PROGRAM MAIN
VAR
END_VAR

TCP_IP();

END_PROGRAM

(* stored: Version 1.1.0.1, ProductVersion 3.1.4024.0
   POU MAIN: Id {8618fe4b-e11c-41e4-a559-71731e97023b}, SpecialFunc None *)
